// TIA Portal V16 export
// export: Created 2025-05-30T16:30:26.912845Z, ExportSetting WithDefaults, DisplayName Totally Integrated Automation Portal, DisplayVersion V16, DisplayName TIA Portal Version Control Interface, DisplayVersion V16, DisplayName TIA Portal Openness, DisplayVersion V16, DisplayName STEP 7 Professional, DisplayVersion V16, DisplayName STEP 7 Safety, DisplayVersion V16, DisplayName WinCC Advanced, DisplayVersion V16
FUNCTION_BLOCK "MC_Jog"   // FB11, FBD
TITLE = MC_Jog
VERSION : 0.1
// With this block you can Jog an Axis manual, you can set the speed on 25%, 50% or 75%. It also has an brake functionality, when you set Brake to true, it holds the brake for 2 seconds, then releases it.
// stored: AutoNumber true, IsIECCheckEnabled false, UDAEnableTagReadback false
   VAR_INPUT
      "Jog Forward" : Bool;
      "Jog Backward" : Bool;
      Speed : Int;
      Brake : Bool;
   END_VAR
   VAR_OUTPUT
      "Drive Fwd Output" : Bool;
      "Drive Rev Output" : Bool;
      "Drive Speed Output" : Int;
      "Drive Brake Output" : Bool;
   END_VAR
BEGIN

REGION Network 1: Manual Control
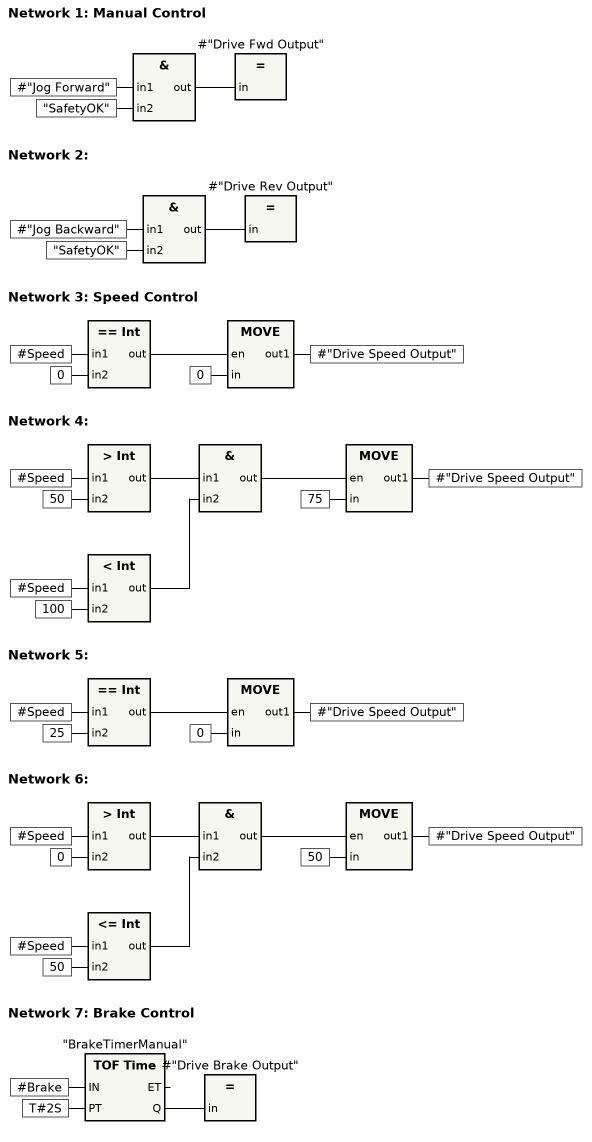
   #"Drive Fwd Output" := #"Jog Forward" AND "SafetyOK";
END_REGION

REGION Network 2
   #"Drive Rev Output" := #"Jog Backward" AND "SafetyOK";
END_REGION

REGION Network 3: Speed Control
   IF #Speed = 0 THEN #"Drive Speed Output" := 0; END_IF;
END_REGION

REGION Network 4
   IF (#Speed > 50) AND (#Speed < 100) THEN #"Drive Speed Output" := 75; END_IF;
END_REGION

REGION Network 5
   IF #Speed = 25 THEN #"Drive Speed Output" := 0; END_IF;
END_REGION

REGION Network 6
   IF (#Speed > 0) AND (#Speed <= 50) THEN #"Drive Speed Output" := 50; END_IF;
END_REGION

REGION Network 7: Brake Control
   "BrakeTimerManual".TOF(IN := #Brake, PT := T#2S);
   #"Drive Brake Output" := "BrakeTimerManual".Q;
END_REGION
END_FUNCTION_BLOCK
